(* CODESYS project codesys_setup.export

Project tree, tasks and I/O mapping:
  libraries: Standard, 3.5.18.0 (System); CmpApp, 3.5.17.0 (System); SysExcept, 3.5.17.0 (System); CmpIecVarAccess, 3.5.17.0 (System); CmpIecTask, * (System); CmpErrors, * (System); SysTypes Interfaces, * (System); CAA Mathematics, * (CAA Technical Workgroup); FloatingPointUtils, 3.5.17.0 (System)
  task CalcFinished (event, event SimulationWatchdog.calculationFinished, priority 2) calls SimulationWatchdog
  task MainTask (cyclic, interval 50 ms, priority 1) calls SimulationWatchdog, PLC_PRG
  data type SimulationState
  program SimulationWatchdog [ST]
*)

// SimulationState
{attribute 'qualified_only'}
{attribute 'strict'}
TYPE SimulationState :
(
	IDLE := 0,
	STEP_TRIGGER := 1,
	STEP_CALCULATION :=2,
	ERROR := 3
);
END_TYPE

// SimulationWatchdog
PROGRAM SimulationWatchdog
VAR_INPUT
	terminate: BOOL;
	run: BOOL := TRUE;
END_VAR
VAR
    //The next two are for getting App instance
    _pApp       : POINTER TO CmpApp.APPLICATION;
    _Result     : SysExcept.SysTypes.RTS_IEC_RESULT;
	
	state: SimulationState := SimulationState.IDLE;
	doStep: BOOL;
	calculationFinished: BOOL;
END_VAR

CASE state OF
	SimulationState.IDLE:
		calculationFinished := FALSE;
		terminate := FALSE;
		doStep := FALSE;
		IF run THEN
			state := SimulationState.STEP_TRIGGER;
		END_IF
		
	SimulationState.STEP_TRIGGER:
		calculationFinished := FALSE;
		IF run THEN
			doStep := TRUE;
			state := SimulationState.STEP_CALCULATION;
		ELSE 
			state := SimulationState.IDLE;
		END_IF
	SimulationState.STEP_CALCULATION:
		IF NOT run THEN
			state := SimulationState.IDLE;
		ELSIF calculationFinished THEN
			doStep := FALSE;
			state := SimulationState.STEP_TRIGGER;
		ELSIF doStep THEN
			state := SimulationState.ERROR;
		END_IF
	SimulationState.ERROR:
		_pApp := AppGetCurrent(pResult := ADR(_Result));
		AppGenerateException(pApp:=_pApp,   ulException:=RtsExceptions.RTSEXCPT_CYCLE_TIME_EXCEED);
END_CASE

END_PROGRAM
